PROGRAM selectPos019
VAR
END_VAR

gvl.cfgPos_OF019:= gvl_p.aPositionsE019[gvl.actPos].numOF;
gvl.cfgPos_LT019:= gvl_p.aPositionsE019[gvl.actPos].lote;
gvl.cfgPos_Class019:= gvl_p.aPositionsE019[gvl.actPos].class;
gvl.cfgPos_Pot019:= gvl_p.aPositionsE019[gvl.actPos].pot;
gvl.cfgPos_Reat019:= gvl_p.aPositionsE019[gvl.actPos].reator;

END_PROGRAM

(* stored: Version 1.1.0.1, ProductVersion 3.1.4024.12
   POU selectPos019: Id {894b9da8-94fd-4354-853e-a18276daef87}, SpecialFunc None *)
